PROGRAM MAIN
VAR
	bStartButton : BOOL; (* Yeşil Başlatma Butonu *)
	bStopButton : BOOL; (* Kırmızı Durdurma Butonu*)
	bMotor : BOOL; (*Çalıştıracağımız Motor*)
END_VAR

IF bStopButton THEN
	bMotor := FALSE;
	
ELSIF bStartButton THEN
	bMotor := TRUE;
END_IF

END_PROGRAM

(* stored: Version 1.1.0.1
   POU MAIN: Id {8b1e4097-6fde-4481-860f-a28426ebbe41}, SpecialFunc None *)
